{attribute 'qualified_only'}
{attribute 'strict'}
{attribute 'to_string'}
TYPE E_1101_Initialization_result : (
		Failure := 0,
		Success := 1
	) UINT;
END_TYPE
//0 - Failure
//	The position initialization can fail for example if
//		- A good position is not found within pos_ini_max_d..-parameters from the given pos init point
//		- A good position is not found within value of pos_init_max_wait_time-parameter
//		- The AGV is not stationary state, it is performing load or there are scanner related errors active.
//1 - Success
//		- A good position was found near the given position initialization point and position was successfully initialized.

(* stored: Version 1.1.0.1, ProductVersion 3.1.4026.17
   DUT E_1101_Initialization_result: Id {fa08dd67-f5bb-4923-984f-76861b9bfca6} *)
